(* CODESYS project Lift Mixed Language.project

Project tree, tasks and I/O mapping:
  Lift : CODESYS Control Win V3, 3S - Smart Software Solutions GmbH, version 3.5.13.20
    application Application
      task Task (cyclic, interval t#20ms, priority 1) calls MainProgramFb, Simulatie
  DeurTest : CODESYS Control Win V3, 3S - Smart Software Solutions GmbH, version 3.5.13.20
    application Application
      task Task (cyclic, interval t#20ms, priority 1) calls DeurTest, Simulatie
  KooiTest : CODESYS Control Win V3, 3S - Smart Software Solutions GmbH, version 3.5.13.20
    application Application
      task Task (cyclic, interval t#20ms, priority 1) calls Simulatie, KooiTest
  Lift Besturing/
    data type DeurToestanden
    data type KooiToestanden
    data type LiftToestanden
    function block KooiFb [ST]
    program MainProgramFb [FBD]
    function block LiftFb [FBD]
    function block BesturingCb [ST]
    function block DeurFb [ST]
    program DeurTest [FBD]
    program KooiTest [FBD]
  global variables GVL
  image pool ImagePool
  5ce3da45-db07-42e7-a21c-a00fff4ed8f6|C:\Users\Gerard\Desktop\MensenInLift.PNG
  5ce3da45-db07-42e7-a21c-a00fff4ed8f6|C:\Users\Gerard\Desktop\LiftDeur.PNG
  5ce3da45-db07-42e7-a21c-a00fff4ed8f6|C:\Users\Gerard\Desktop\Liftaandrijving.PNG
  5ce3da45-db07-42e7-a21c-a00fff4ed8f6|C:\Users\Gerard\Desktop\LiftDeurAandrijving.PNG
  Lift Simualtie/
    program Simulatie [ST]
  text list GlobalTextList
  visualisation Visualization
*)

// Lift Besturing/DeurToestanden
// Authour : G A Harkema
// Date:  february 15, 2017
// Version : 1.0
// States of the door
TYPE DeurToestanden :
(
	idle := 0,close, toOpen, open, toClose
);
END_TYPE

// Lift Besturing/KooiToestanden
// Authour : G A Harkema
// Date:  february 15, 2017
// Version : 1.0
// States of the cage
TYPE KooiToestanden :
(
	idle := 0, stationary, goUp, goDown  
);
END_TYPE

// Lift Besturing/LiftToestanden
// Authour : G A Harkema
// Date:  february 15, 2017
// Version : 1.0
// States of the cage
TYPE LiftToestanden :
(
	idle := 0, waitForChoise, closingDoor, preTraveling, traveling, openingDoor
);
END_TYPE

// GVL
VAR_GLOBAL
	Ix_BovenOproepKooi					: BOOL;
	Ix_BenedenOproepKooi				: BOOL;
	Ix_KooiGaNaarBoven					: BOOL;
	Ix_KooiGaNaarBeneden				: BOOL;
	Ix_KooiBoven						: BOOL;
	Ix_KooiBeneden						: BOOL;
	Qx_AandrijvingOmhoog				: BOOL;
	Qx_AandrijvingOmlaag				: BOOL;
	
	
	Ix_BenedenDeurOpen					: BOOL;
	Ix_BenedenDeurGesloten				: BOOL;
	Qx_BenedenDeurAandrijvingOpen		: BOOL;
	Qx_BenedenDeurAandrijvingSluiten	: BOOL;
	
	Ix_BovenDeurOpen					: BOOL;
	Ix_BovenDeurGesloten				: BOOL;
	Qx_BovenDeurAandrijvingOpen			: BOOL;
	Qx_BovenDeurAandrijvingSluiten		: BOOL;
	
	Ix_TestButton1						: BOOL;
	Ix_TestButton2						: BOOL;
	Ix_TestButton3						: BOOL;
	
	Qx_TestIndicator1					: BOOL;
	Qx_TestIndicator2					: BOOL;
	Qx_TestIndicator3					: BOOL;
	
END_VAR

// Lift Besturing/MainProgramFb
PROGRAM MainProgramFb
VAR
	Lift: LiftFb;
END_VAR

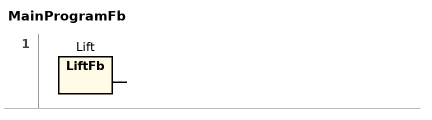
// NETWORK 1
Lift(); // LiftFb

END_PROGRAM

// Lift Besturing/LiftFb
FUNCTION_BLOCK LiftFb
VAR
	DeurBenden					: DeurFb;
	Besturing					: BesturingCb;
	DeurBoven					: DeurFb;
	Kooi						: KooiFb;
	KooiBoven					: BOOL;
	DeurBovenIsOpen				: BOOL;
	DeurBenedenIsOpen			: BOOL;
	DeurBovenIsGesloten			: BOOL;
	DeurBenedenIsGesloten		: BOOL;
	DeurBenedenGaOpen			: BOOL;
	DeurBenedenGaSluiten		: BOOL;
	DeurBovenGaOpen				: BOOL;
	DeurBovenGaSluiten			: BOOL;
	KooiBeneden					: BOOL;
	KooiStart					: BOOL;
END_VAR

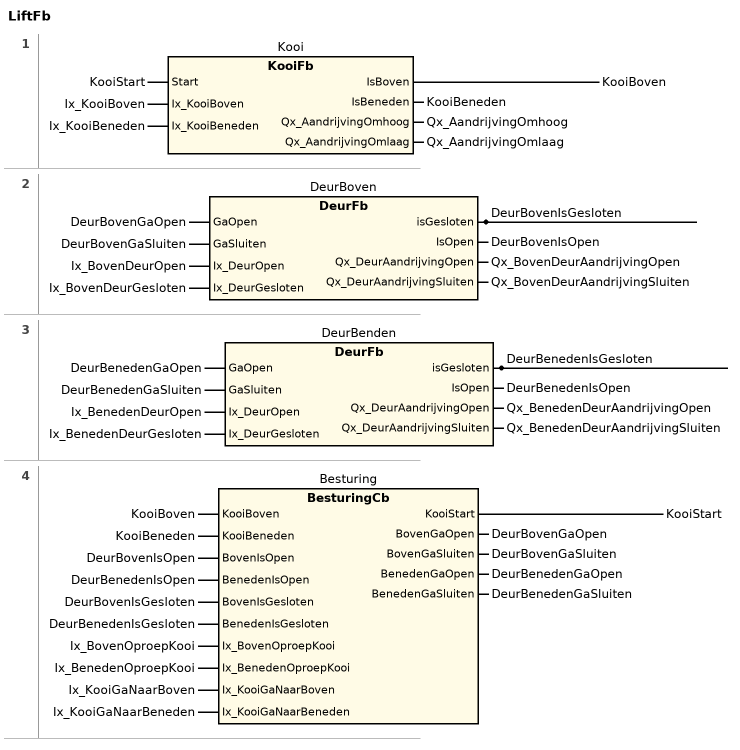
// NETWORK 1
Kooi(
    Start := KooiStart,
    Ix_KooiBoven := Ix_KooiBoven,
    Ix_KooiBeneden := Ix_KooiBeneden,
    IsBeneden => KooiBeneden,
    Qx_AandrijvingOmhoog => Qx_AandrijvingOmhoog,
    Qx_AandrijvingOmlaag => Qx_AandrijvingOmlaag); // KooiFb
KooiBoven := Kooi.IsBoven;

// NETWORK 2
DeurBoven(
    GaOpen := DeurBovenGaOpen,
    GaSluiten := DeurBovenGaSluiten,
    Ix_DeurOpen := Ix_BovenDeurOpen,
    Ix_DeurGesloten := Ix_BovenDeurGesloten,
    isGesloten => DeurBovenIsGesloten,
    IsOpen => DeurBovenIsOpen,
    Qx_DeurAandrijvingOpen => Qx_BovenDeurAandrijvingOpen,
    Qx_DeurAandrijvingSluiten => Qx_BovenDeurAandrijvingSluiten); // DeurFb

// NETWORK 3
DeurBenden(
    GaOpen := DeurBenedenGaOpen,
    GaSluiten := DeurBenedenGaSluiten,
    Ix_DeurOpen := Ix_BenedenDeurOpen,
    Ix_DeurGesloten := Ix_BenedenDeurGesloten,
    isGesloten => DeurBenedenIsGesloten,
    IsOpen => DeurBenedenIsOpen,
    Qx_DeurAandrijvingOpen => Qx_BenedenDeurAandrijvingOpen,
    Qx_DeurAandrijvingSluiten => Qx_BenedenDeurAandrijvingSluiten); // DeurFb

// NETWORK 4
Besturing(
    KooiBoven := KooiBoven,
    KooiBeneden := KooiBeneden,
    BovenIsOpen := DeurBovenIsOpen,
    BenedenIsOpen := DeurBenedenIsOpen,
    BovenIsGesloten := DeurBovenIsGesloten,
    BenedenIsGesloten := DeurBenedenIsGesloten,
    Ix_BovenOproepKooi := Ix_BovenOproepKooi,
    Ix_BenedenOproepKooi := Ix_BenedenOproepKooi,
    Ix_KooiGaNaarBoven := Ix_KooiGaNaarBoven,
    Ix_KooiGaNaarBeneden := Ix_KooiGaNaarBeneden,
    BovenGaOpen => DeurBovenGaOpen,
    BovenGaSluiten => DeurBovenGaSluiten,
    BenedenGaOpen => DeurBenedenGaOpen,
    BenedenGaSluiten => DeurBenedenGaSluiten); // BesturingCb
KooiStart := Besturing.KooiStart;

END_FUNCTION_BLOCK

// Lift Besturing/KooiFb
FUNCTION_BLOCK KooiFb
VAR_INPUT
	Start 								: BOOL;

	Ix_KooiBoven						: BOOL;
	Ix_KooiBeneden						: BOOL;
END_VAR

VAR_OUTPUT
	IsBoven								: BOOL;
	IsBeneden							: BOOL;

	Qx_AandrijvingOmhoog				: BOOL;
	Qx_AandrijvingOmlaag				: BOOL;
END_VAR

VAR
	Toestand							: KooiToestanden := KooiToestanden.idle;
	initialiazed 						: BOOL := FALSE;
END_VAR

IF NOT initialiazed THEN
// Set default values
	Qx_AandrijvingOmhoog 	:= FALSE;
	Qx_AandrijvingOmlaag 	:= FALSE;

	initialiazed := TRUE;
END_IF


CASE Toestand OF
	KooiToestanden.idle:
		Qx_AandrijvingOmlaag := TRUE;  // powerup sequence
		Toestand := KooiToestanden.goDown;

	KooiToestanden.goDown:
		IF Ix_KooiBeneden THEN  // Handle downstair event
			Qx_AandrijvingOmlaag := FALSE;
			Toestand := KooiToestanden.stationary;
		END_IF
	
	KooiToestanden.goUp:
		IF Ix_KooiBoven THEN  // Handle upstairs event
			Qx_AandrijvingOmhoog := FALSE;
			Toestand := KooiToestanden.stationary;
		END_IF
END_CASE

IF Start THEN
	IF Toestand = KooiToestanden.stationary THEN
		
		// Check position of the cage and handle
		IF IsBoven THEN
			Qx_AandrijvingOmlaag := TRUE;
			Toestand := KooiToestanden.goDown;
		END_IF
		
		IF IsBeneden THEN
			Qx_AandrijvingOmhoog := TRUE;
			Toestand := KooiToestanden.goUp;
		END_IF
	END_IF
END_IF

IsBoven := Ix_KooiBoven;
IsBeneden := Ix_KooiBeneden;

END_FUNCTION_BLOCK

// Lift Besturing/DeurFb
FUNCTION_BLOCK DeurFb
VAR_INPUT
	GaOpen						: BOOL;
	GaSluiten					: BOOL;

	Ix_DeurOpen					: BOOL;
	Ix_DeurGesloten				: BOOL;
END_VAR
VAR_OUTPUT
	isGesloten					: BOOL;			
	IsOpen						: BOOL;

	Qx_DeurAandrijvingOpen		: BOOL;
	Qx_DeurAandrijvingSluiten	: BOOL;
END_VAR

VAR
	Toestand						: DeurToestanden := DeurToestanden.idle;
	initialiazed 				: BOOL := FALSE;
	eState: DeurToestanden;
END_VAR

IF NOT initialiazed THEN
	Qx_DeurAandrijvingOpen := FALSE;
	Qx_DeurAandrijvingSluiten := TRUE;
	// Trigger door when close
	IF Toestand = DeurToestanden.idle THEN
		Toestand := DeurToestanden.toClose; // Hnadle event
		Qx_DeurAandrijvingSluiten := TRUE;
	END_IF
	initialiazed := TRUE;
END_IF

CASE Toestand OF
	DeurToestanden.toOpen :
		IF Ix_DeurOpen THEN  // handle open event
			Qx_DeurAandrijvingOpen := FALSE;
			Toestand := DeurToestanden.open;
		END_IF
	
	DeurToestanden.toClose :
		IF Ix_DeurGesloten THEN // handle close event
			Qx_DeurAandrijvingSluiten := FALSE;
			Toestand := DeurToestanden.close;
		END_IF
	
END_CASE


IF GaOpen THEN
	IF Toestand = DeurToestanden.close THEN
		Toestand := DeurToestanden.toOpen;  // Handle event
		Qx_DeurAandrijvingOpen := TRUE;
	END_IF
END_IF


// Trigger door when close
IF GaSluiten THEN
	IF Toestand = DeurToestanden.Open THEN
		Toestand := DeurToestanden.toClose; // Hnadle event
		Qx_DeurAandrijvingSluiten := TRUE;
	END_IF
END_IF

isGesloten := Toestand = DeurToestanden.close;
isOpen := Toestand = DeurToestanden.open;

END_FUNCTION_BLOCK

// Lift Besturing/BesturingCb
FUNCTION_BLOCK BesturingCb
VAR_INPUT
	KooiBoven						: BOOL;
	KooiBeneden						: BOOL;

	BovenIsOpen						: BOOL;
	BenedenIsOpen					: BOOL;			
	BovenIsGesloten					: BOOL;
	BenedenIsGesloten				: BOOL;			
	
	Ix_BovenOproepKooi				: BOOL;
	Ix_BenedenOproepKooi			: BOOL;
	Ix_KooiGaNaarBoven				: BOOL;
	Ix_KooiGaNaarBeneden			: BOOL;
END_VAR

VAR_OUTPUT
	KooiStart						: BOOL;
	
	BovenGaOpen						: BOOL;
	BovenGaSluiten					: BOOL;
	BenedenGaOpen					: BOOL;
	BenedenGaSluiten				: BOOL;
END_VAR

VAR
	initialiazed	 				: BOOL := FALSE;
	Toestand						: LiftToestanden := LiftToestanden.idle;
END_VAR

IF NOT initialiazed THEN
	initialiazed := TRUE;
END_IF


CASE Toestand OF
	LiftToestanden.idle:
		Toestand := LiftToestanden.waitForChoise;

	LiftToestanden.waitForChoise:
		IF KooiBoven THEN  // welke keuze
			IF Ix_KooiGaNaarBeneden OR Ix_BenedenOproepKooi THEN
				BovenGaSluiten := TRUE; // Creeer event
				Toestand := LiftToestanden.closingDoor;
			END_IF
		END_IF
		
		IF KooiBeneden THEN // welke keuze
			IF Ix_KooiGaNaarBoven OR Ix_BovenOproepKooi THEN
				BenedenGaSluiten := TRUE; // Creeer event
				Toestand := LiftToestanden.closingDoor;
			END_IF
		END_IF

	LiftToestanden.closingDoor:
		BenedenGaSluiten := FALSE; // verwijder event
		BovenGaSluiten := FALSE; // verwijder event
		IF BovenIsGesloten AND BenedenIsGesloten THEN // handle doors closed
			KooiStart := TRUE;
			Toestand := LiftToestanden.PreTraveling;
		END_IF
		
	LiftToestanden.preTraveling: // wachten op het starten van het reizen van de kooi
		IF NOT (KooiBoven OR KooiBeneden) THEN
			Toestand := LiftToestanden.Traveling;
			KooiStart := FALSE; // verwijder event
		END_IF 
		
	LiftToestanden.traveling:
		IF (KooiBoven OR KooiBeneden) THEN // handle arriving of cage
			IF KooiBoven  THEN
				BovenGaOpen := TRUE; // Creeer event
				Toestand := LiftToestanden.openingDoor;
			END_IF
	
			IF KooiBeneden THEN
				BenedenGaOpen := TRUE; // Creeer event
				Toestand := LiftToestanden.openingDoor;
			END_IF
		END_IF;

	LiftToestanden.openingDoor:
		BovenGaOpen := FALSE; // verwijder event
		BenedenGaOpen := FALSE; // verwijder event
		IF BovenIsOpen OR BenedenIsOpen THEN // Handle door open
			Toestand := LiftToestanden.waitForChoise;
		END_IF
END_CASE

END_FUNCTION_BLOCK

// Lift Simualtie/Simulatie
// Programma		: Simulatie
// Project			: Lift
// Doel				: Simulatie functies voor de lift
// Auteur			: Gerard Harkema
// Versie			: 1.0
// Datum			: 15 oktober 2015

PROGRAM Simulatie
VAR

	Mw_PositieLiftInv					: INT := 0;
	Mw_PositieLift						: INT := 0;
	Mw_LiftBenedenCountValue			: INT := 250;

	Mw_BenedenPositieDeur				: INT := 0;
	Mw_BenedenPositieDeurCountValue		: INT := 100;

	Mw_BovenPositieDeur					: INT := 0;
	Mw_BovenPositieDeurCountValue		: INT := 100;

END_VAR


// Reizen lift omhoog
IF(GVL.Qx_AandrijvingOmhoog AND (NOT GVL.Ix_KooiBoven)) THEN
	Mw_PositieLiftInv := Mw_PositieLiftInv + 1;
END_IF

// Reizen lift omlaag
IF(GVL.Qx_AandrijvingOmlaag AND (NOT GVL.Ix_KooiBeneden)) THEN
	Mw_PositieLiftInv := Mw_PositieLiftInv - 1;
END_IF

Mw_PositieLift := Mw_LiftBenedenCountValue - Mw_PositieLiftInv;

// Detectie lift is boven
IF (Mw_PositieLiftInv >= Mw_LiftBenedenCountValue) THEN
	GVL.Ix_KooiBoven := TRUE;
ELSE
	GVL.Ix_KooiBoven := FALSE;	
END_IF
  

// Detectie lift is beneden
IF(Mw_PositieLiftInv <= 0) THEN
	GVL.Ix_KooiBeneden := TRUE;
ELSE
	GVL.Ix_KooiBeneden := FALSE;	
END_IF

// Inactief maken oproepknoppen
IF GVL.Ix_KooiBoven THEN
 Ix_BovenOproepKooi := FALSE;
 Ix_KooiGaNaarBoven := FALSE;
END_IF

IF GVL.Ix_KooiBeneden THEN
 Ix_BenedenOproepKooi := FALSE;
 Ix_KooiGaNaarBeneden := FALSE;
END_IF


//*********************************************
//                 Bovendeur
//*********************************************

// Bovendeur openen
IF(GVL.Qx_BovenDeurAandrijvingOpen AND (NOT GVL.Ix_BovenDeurOpen)) THEN
	Mw_BovenPositieDeur := Mw_BovenPositieDeur + 1;
END_IF

// Bovendeur sluiten
IF(GVL.Qx_BovenDeurAandrijvingSluiten AND (NOT GVL.Ix_BovenDeurGesloten)) THEN
	Mw_BovenPositieDeur := Mw_BovenPositieDeur - 1;
END_IF

IF (Mw_BovenPositieDeur >= Mw_BovenPositieDeurCountValue) THEN
	GVL.Ix_BovenDeurOpen := TRUE;
ELSE
	GVL.Ix_BovenDeurOpen := FALSE;	
END_IF
  

// Detectie bovendeur is gesloten
IF(Mw_BovenPositieDeur <= 0) THEN
	GVL.Ix_BovenDeurGesloten := TRUE;
ELSE
	GVL.Ix_BovenDeurGesloten := FALSE;	
END_IF

//*********************************************
//                 Benedendeur
//*********************************************

// Benedendeur openen
IF(GVL.Qx_BenedenDeurAandrijvingOpen AND (NOT GVL.Ix_BenedenDeurOpen)) THEN
	Mw_BenedenPositieDeur := Mw_BenedenPositieDeur + 1;
END_IF

// Benedendeur sluiten
IF(GVL.Qx_BenedenDeurAandrijvingSluiten AND (NOT GVL.Ix_BenedenDeurGesloten)) THEN
	Mw_BenedenPositieDeur := Mw_BenedenPositieDeur - 1;
END_IF

// Detectie Benedendeur is open
IF (Mw_BenedenPositieDeur >= Mw_BenedenPositieDeurCountValue) THEN
	GVL.Ix_BenedenDeurOpen := TRUE;
ELSE
	GVL.Ix_BenedenDeurOpen := FALSE;	
END_IF

// Detectie Benedendeur is gesloten
IF(Mw_BenedenPositieDeur <= 0) THEN
	GVL.Ix_BenedenDeurGesloten := TRUE;
ELSE
	GVL.Ix_BenedenDeurGesloten := FALSE;	
END_IF

END_PROGRAM

// Lift Besturing/DeurTest
PROGRAM DeurTest
VAR
	DeurBoven: DeurFb;
END_VAR

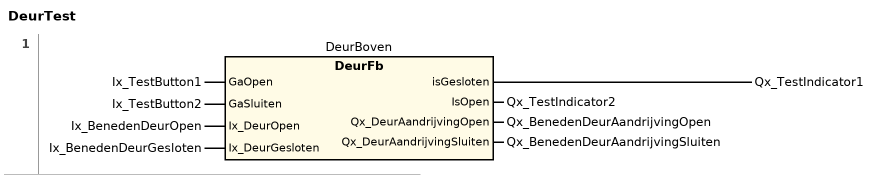
// NETWORK 1
DeurBoven(
    GaOpen := Ix_TestButton1,
    GaSluiten := Ix_TestButton2,
    Ix_DeurOpen := Ix_BenedenDeurOpen,
    Ix_DeurGesloten := Ix_BenedenDeurGesloten,
    IsOpen => Qx_TestIndicator2,
    Qx_DeurAandrijvingOpen => Qx_BenedenDeurAandrijvingOpen,
    Qx_DeurAandrijvingSluiten => Qx_BenedenDeurAandrijvingSluiten); // DeurFb
Qx_TestIndicator1 := DeurBoven.isGesloten;

END_PROGRAM

// Lift Besturing/KooiTest
PROGRAM KooiTest
VAR
	Kooi: KooiFb;
END_VAR

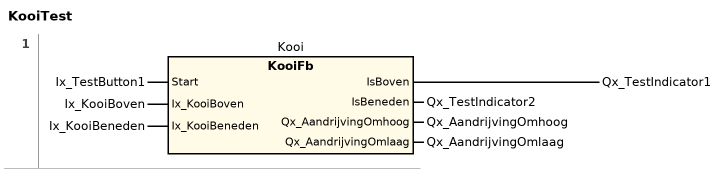
// NETWORK 1
Kooi(
    Start := Ix_TestButton1,
    Ix_KooiBoven := Ix_KooiBoven,
    Ix_KooiBeneden := Ix_KooiBeneden,
    IsBeneden => Qx_TestIndicator2,
    Qx_AandrijvingOmhoog => Qx_AandrijvingOmhoog,
    Qx_AandrijvingOmlaag => Qx_AandrijvingOmlaag); // KooiFb
Qx_TestIndicator1 := Kooi.IsBoven;

END_PROGRAM

// /Visualization
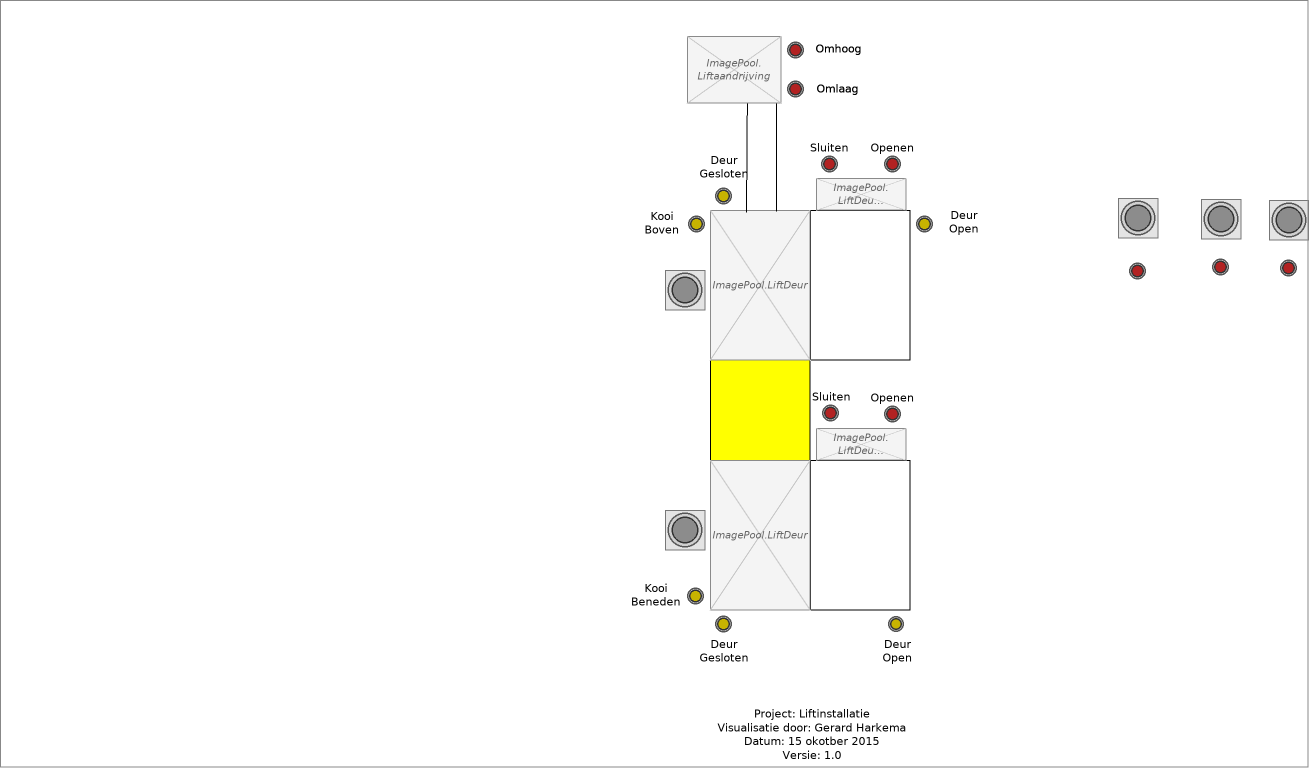
VISUALIZATION Visualization  // 1309x768
    Rectangle (810,460 100x150)
    Rectangle (810,210 100x150)
    Rectangle (710,210 100x400)
    PushSwitch (665,270 40x40), tooltip "Oproep Boven", variable: Ix_BovenOproepKooi, behaviour: TOGGLE, style: Switch-PushSwitch-Gray
    PushSwitch (665,510 40x40), tooltip "Oproep Beneden", variable: Ix_BenedenOproepKooi, behaviour: TOGGLE, style: Switch-PushSwitch-Gray
    Group (710,210 100x150)
        p2738717112: Simulatie.Mw_PositieLift
        Rectangle (0,0 100x150)
        Image (6,0 89x150), image: ImagePool.MensenInLift
        PushSwitch (5,100 30x30), tooltip "Ga naar beneden", variable: Ix_KooiGaNaarBeneden, behaviour: TOGGLE, style: Switch-PushSwitch-Gray
        PushSwitch (5,60 30x30), tooltip "Ga naar Boven", variable: Ix_KooiGaNaarBoven, behaviour: TOGGLE, style: Switch-PushSwitch-Gray
    Rectangle (710,210 100x150)
    Image (716,210 89x150), image: ImagePool.MensenInLift
    PushSwitch (715,310 30x30), tooltip "Ga naar beneden", variable: Ix_KooiGaNaarBeneden, behaviour: TOGGLE, style: Switch-PushSwitch-Gray
    PushSwitch (715,270 30x30), tooltip "Ga naar Boven", variable: Ix_KooiGaNaarBoven, behaviour: TOGGLE, style: Switch-PushSwitch-Gray
    Lamp1 (714,186 19x20), variable: Ix_BovenDeurGesloten, style: Lamp-Lamp1-Yellow
    Lamp1 (915,214 19x20), variable: Ix_BovenDeurOpen, style: Lamp-Lamp1-Yellow
    Lamp1 (687,214 19x20), variable: Ix_KooiBoven, style: Lamp-Lamp1-Yellow
    Lamp1 (686,586 19x20), variable: Ix_KooiBeneden, style: Lamp-Lamp1-Yellow
    Lamp1 (714,614 19x20), variable: Ix_BenedenDeurGesloten, style: Lamp-Lamp1-Yellow
    Lamp1 (887,614 18x20), variable: Ix_BenedenDeurOpen, style: Lamp-Lamp1-Yellow
    Label (682,152 84x30), "Deur Gesloten"
    Label (937,207 54x30), "Deur Open"
    Label (640,208 44x30), "Kooi Boven"
    Label (629,580 54x30), "Kooi Beneden"
    Label (693,636 62x30), "Deur Gesloten"
    Label (875,636 45x30), "Deur Open"
    Group (710,210 100x150)
        p3560616238: Simulatie.Mw_BovenPositieDeur
        Rectangle (0,0 100x150)
        Image (0,0 100x150), image: ImagePool.LiftDeur
    Group (710,460 100x150)
        p3560616238: Simulatie.Mw_BenedenPositieDeur
        Rectangle (0,0 100x150)
        Image (0,0 100x150), image: ImagePool.LiftDeur
    Line (747,83) (746,212)
    Line (776,82) (776,211)
    Group (687,34 182x70)
        Image (0,2 94x67), image: ImagePool.Liftaandrijving
        Lamp1 (99,6 19x20), variable: Qx_AandrijvingOmhoog, style: Lamp-Lamp1-Red
        Lamp1 (99,45 19x20), variable: Qx_AandrijvingOmlaag, style: Lamp-Lamp1-Red
        Label (121,0 61x30), "Omhoog"
        Label (123,40 55x30), "Omlaag"
    Image (687,36 94x67), image: ImagePool.Liftaandrijving
    Lamp1 (786,40 19x20), variable: Qx_AandrijvingOmhoog, style: Lamp-Lamp1-Red
    Lamp1 (786,79 19x20), variable: Qx_AandrijvingOmlaag, style: Lamp-Lamp1-Red
    Label (808,34 61x30), "Omhoog"
    Label (810,74 55x30), "Omlaag"
    Group (816,154 90x56)
        Image (0,24 90x32), image: ImagePool.LiftDeurAandrijving
        Lamp1 (4,0 19x20), variable: Qx_BovenDeurAandrijvingSluiten, style: Lamp-Lamp1-Red
        Lamp1 (67,0 19x20), variable: Qx_BovenDeurAandrijvingOpen, style: Lamp-Lamp1-Red
    Image (816,178 90x32), image: ImagePool.LiftDeurAandrijving
    Lamp1 (820,154 19x20), variable: Qx_BovenDeurAandrijvingSluiten, style: Lamp-Lamp1-Red
    Lamp1 (883,154 19x20), variable: Qx_BovenDeurAandrijvingOpen, style: Lamp-Lamp1-Red
    Group (816,403 90x57)
        Image (0,25 90x32), image: ImagePool.LiftDeurAandrijving
        Lamp1 (5,0 19x20), variable: Qx_BenedenDeurAandrijvingSluiten, style: Lamp-Lamp1-Red
        Lamp1 (67,1 19x20), variable: Qx_BenedenDeurAandrijvingOpen, style: Lamp-Lamp1-Red
    Image (816,428 90x32), image: ImagePool.LiftDeurAandrijving
    Lamp1 (821,403 19x20), variable: Qx_BenedenDeurAandrijvingSluiten, style: Lamp-Lamp1-Red
    Lamp1 (883,404 19x20), variable: Qx_BenedenDeurAandrijvingOpen, style: Lamp-Lamp1-Red
    Label (812,382 39x30), "Sluiten"
    Label (810,133 39x30), "Sluiten"
    Label (867,383 51x30), "Openen"
    Label (867,133 51x30), "Openen"
    Label (712,701 200x67), "Project: Liftinstallatie Visualisatie door: Gerard Harkema Datum: 15 okotber 2015 Versie: 1.0"
    PushSwitch (1118,198 40x40), tooltip "Test Button 1", variable: Ix_TestButton1, behaviour: TOGGLE, style: Switch-PushSwitch-Gray
    PushSwitch (1201,199 40x40), tooltip "Test Button 2", variable: Ix_TestButton2, behaviour: TOGGLE, style: Switch-PushSwitch-Gray
    Lamp1 (1128,261 19x20), variable: Qx_TestIndicator1, style: Lamp-Lamp1-Red
    Lamp1 (1211,257 19x20), variable: Qx_TestIndicator2, style: Lamp-Lamp1-Red
    PushSwitch (1269,200 40x40), tooltip "Test Button 2", variable: Ix_TestButton3, behaviour: TOGGLE, style: Switch-PushSwitch-Gray
    Lamp1 (1279,258 19x20), variable: Qx_TestIndicator3, style: Lamp-Lamp1-Red
END_VISUALIZATION
